TYPE ST_GenGridController_SyncData :
STRUCT
	b_Sync				: BOOL;
	r_freqSet			: REAL;
	r_VoltSet			: REAL;
END_STRUCT
END_TYPE

(* stored: Version 1.1.0.1, ProductVersion 3.1.4026.18
   DUT ST_GenGridController_SyncData: Id {1e1e58db-cc8b-42fb-b865-94dc18038922} *)
